RoboDK station: M20_v48.rdk

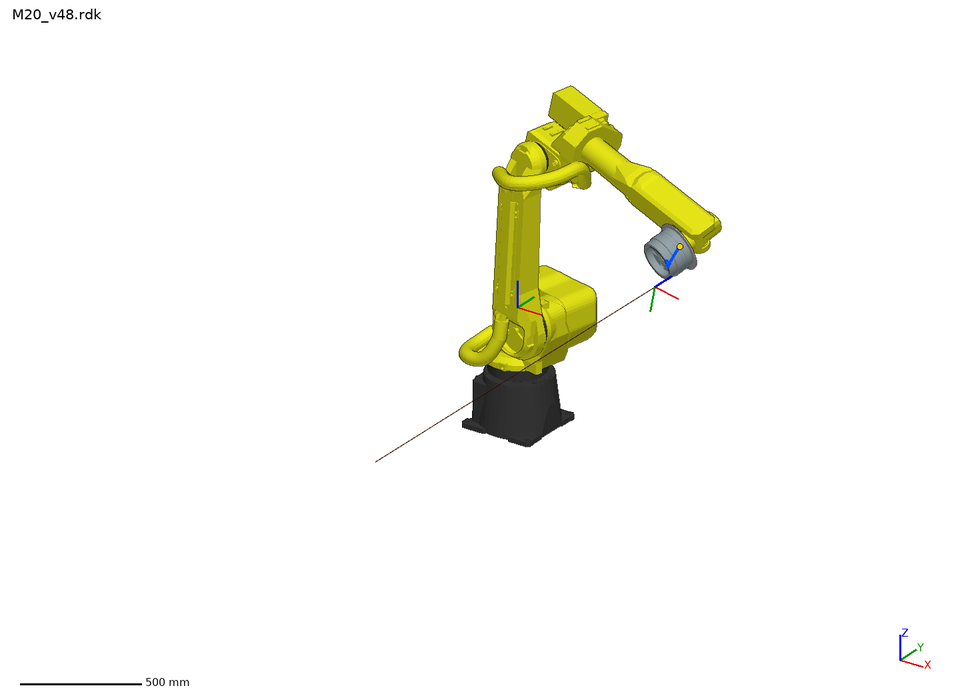
[picture v0: the station drawn from its stored meshes, robots at their saved joint values, targets as dots, program paths as lines]
Station M20_v48 (saved by RoboDK 5.2.2). Poses are relative to the parent item; angles as X-Y-Z fixed-axis rotations.
Station parameters (name, value as stored): CollisionFreePlanner, Fanuc M-20iA/35M, CollisionFreePlanner-Rob Fanuc M-20iA/35M
  - frame Fanuc M-20iA/35M Base at (0, 0, 525) mm
    - frame LASER_RTCP at (1000.3, -445, 552.3) mm, rotated rx -90 ry 10.19 rz 0 deg
      - object LASER_CAD at (0, 0, -1005) mm, size 2 x 2 x 2000 mm, geometry from laser.stl
    - robot Fanuc M-20iA/35M: 6 axes, payload 35 kg, reach 1813 mm, repeatability 0.04 mm, weight 252 kg
        modified DH rows (alpha deg, a mm, theta deg, d mm): 0, 0, 0, 525; -90, 150, -90, 0; 0, 790, 0, 0; -90, 150, 0, 860; 90, 0, 0, 0; -90, 0, 0, 100
        base shift (0, 0, -525) mm
        joint limits [-185, -110, -85, -200, -190, -450] to [185, 110, 245, 200, 190, 450]; home [0, 0, 0, 0, 0, 0]; saved at [-11.342, 3.915, -14.311, 70.129, -92.08, -387.18]
      - tool DIECAST, TCP at (0, 0, 200) mm, size 185 x 185 x 115 mm, geometry from B2 62-24 3naka.stp
      - tool Diecast15, TCP at (0, 0, 0) mm, geometry from I Co
      - tool holder_cylinder, TCP at (0, 0, 200) mm, size 220 x 220 x 5 mm, geometry from holder_cylinder.stl
  - machining project Diecast15 Settings: rotZ(0) | rotX(0)*rotY(0) | onStart | onPathStart | onApproach | onPoint | onRetract | onFinish | SetRPM(%1) | SetTool(%1) | Extruder(%1) | default | default | OutOnMov(%1) | OutOffMov(%1) | onPathFinish | M_RunCode(%1)
  - program Diecast15 (465 instructions, listed below)
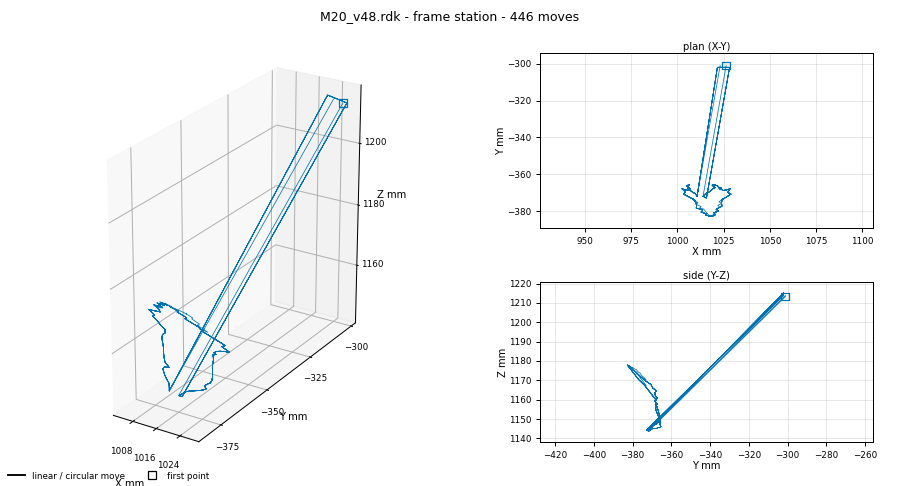
[picture p0: tool path of M20_v48.rdk in frame station, 446 of 446 moves have a stored position in this frame; points joined in program order, loops and branches not executed]

--- program Diecast15 (robot Fanuc M-20iA/35M) ---
  Smooth(1)
  Set speed (50.0 mm/s)
  Set Ref.: LASER_RTCP
  Set Tool: Diecast15
  Show Diecast15
  MoveJ 1 to (1.63, -138.5, 143.91) mm, rotated rx -165.35 ry -21.88 rz 21.81 deg; joints [-11.825, 0.745, -13.905, 69.881, -63.946, 28.2]
  MoveL 2 to (1.63, -138.5, 143.91) mm, rotated rx -165.35 ry -21.88 rz 21.81 deg; joints [-11.825, 0.745, -13.905, 69.881, -63.946, 28.2]
  MoveL 3 to (1.63, -67.79, 73.2) mm, rotated rx -165.35 ry -21.88 rz 21.81 deg; joints [-15.798, 1.644, -18.484, 72.688, -58.86, 24.658]
  MoveL 4 to (1.63, -67.79, 73.2) mm, rotated rx -165.35 ry -21.88 rz 21.81 deg; joints [-15.798, 1.644, -18.484, 72.688, -58.86, 24.658]
  Set speed (10.0 mm/s)
  MoveL 5 to (2.07, -68.2, 73.76) mm, rotated rx -165.47 ry -21.99 rz 21.64 deg; joints [-15.768, 1.64, -18.47, 72.794, -58.687, 24.483]
  MoveL 6 to (2.53, -68.64, 74.3) mm, rotated rx -165.57 ry -22.1 rz 21.49 deg; joints [-15.738, 1.639, -18.452, 72.873, -58.521, 24.337]
  MoveL 7 to (3.06, -69.11, 74.82) mm, rotated rx -165.64 ry -22.21 rz 21.37 deg; joints [-15.708, 1.647, -18.431, 72.918, -58.387, 24.236]
  MoveL 8 to (4.19, -69.63, 75.26) mm, rotated rx -165.57 ry -22.14 rz 21.47 deg; joints [-15.663, 1.734, -18.403, 72.823, -58.562, 24.363]
  MoveL 9 to (5.25, -69.87, 75.97) mm, rotated rx -165.69 ry -21.9 rz 21.48 deg; joints [-15.595, 1.808, -18.422, 73.065, -58.781, 24.144]
  MoveL 10 to (6.16, -70.02, 76.76) mm, rotated rx -165.89 ry -21.66 rz 21.42 deg; joints [-15.526, 1.864, -18.454, 73.413, -58.948, 23.797]
  MoveL 11 to (6.84, -70.15, 77.58) mm, rotated rx -166.69 ry -23.17 rz 23.41 deg; joints [-15.529, 1.8, -18.399, 72.916, -58.015, 26.249]
  MoveL 12 to (7.69, -70.84, 77.79) mm, rotated rx -166.55 ry -23.35 rz 23.41 deg; joints [-15.514, 1.85, -18.34, 72.636, -57.944, 26.482]
  MoveL 13 to (6.15, -70.44, 79.2) mm, rotated rx -167.55 ry -23.65 rz 22.5 deg; joints [-15.485, 1.581, -18.448, 73.906, -56.916, 24.951]
  MoveL 14 to (6.63, -71.02, 79.57) mm, rotated rx -167.55 ry -23.88 rz 22.37 deg; joints [-15.471, 1.583, -18.407, 73.817, -56.696, 24.96]
  MoveL 15 to (7.97, -72.41, 79.13) mm, rotated rx -166.89 ry -24.33 rz 22.62 deg; joints [-15.496, 1.704, -18.238, 72.683, -56.704, 26.052]
  MoveL 16 to (8.34, -73.51, 79.04) mm, rotated rx -166.59 ry -24.9 rz 22.52 deg; joints [-15.528, 1.7, -18.115, 72.031, -56.302, 26.565]
  MoveL 17 to (8.5, -74.86, 78.73) mm, rotated rx -166.17 ry -25.7 rz 22.39 deg; joints [-15.588, 1.674, -17.952, 71.101, -55.743, 27.309]
  MoveL 18 to (8.44, -76.15, 78.49) mm, rotated rx -166.38 ry -28.16 rz 24.17 deg; joints [-15.723, 1.552, -17.704, 69.121, -54.238, 30.819]
  MoveL 19 to (8.5, -77.42, 78.01) mm, rotated rx -165.94 ry -28.95 rz 23.91 deg; joints [-15.798, 1.526, -17.548, 68.152, -53.692, 31.516]
  MoveL 20 to (8.57, -78.66, 77.54) mm, rotated rx -165.5 ry -29.73 rz 23.67 deg; joints [-15.871, 1.503, -17.397, 67.191, -53.168, 32.216]
  MoveL 21 to (8.69, -79.8, 77.16) mm, rotated rx -165.12 ry -30.43 rz 23.43 deg; joints [-15.935, 1.485, -17.262, 66.331, -52.694, 32.845]
  MoveL 22 to (8.83, -80.8, 76.93) mm, rotated rx -164.84 ry -31.04 rz 23.21 deg; joints [-15.986, 1.466, -17.149, 65.628, -52.254, 33.35]
  MoveL 23 to (8.86, -81.65, 76.86) mm, rotated rx -164.67 ry -31.59 rz 22.95 deg; joints [-16.027, 1.43, -17.059, 65.109, -51.784, 33.692]
  MoveL 24 to (8.62, -82.36, 76.99) mm, rotated rx -164.65 ry -32.12 rz 22.64 deg; joints [-16.061, 1.358, -16.994, 64.807, -51.211, 33.829]
  MoveL 25 to (8.14, -82.88, 77.34) mm, rotated rx -164.81 ry -32.62 rz 22.28 deg; joints [-16.085, 1.251, -16.958, 64.762, -50.545, 33.726]
  MoveL 26 to (8.9, -83.1, 77.88) mm, rotated rx -164.95 ry -32.61 rz 22.32 deg; joints [-16.042, 1.287, -16.962, 64.907, -50.532, 33.64]
  MoveL 27 to (8.4, -83.82, 77.16) mm, rotated rx -163.11 ry -28.11 rz 16.62 deg; joints [-15.881, 1.436, -17.144, 68.063, -52.662, 25.505]
  MoveL 28 to (9.59, -85.18, 76.37) mm, rotated rx -162.32 ry -28.55 rz 16.51 deg; joints [-15.938, 1.548, -16.98, 66.869, -52.596, 26.417]
  MoveL 29 to (10.68, -85.68, 76.53) mm, rotated rx -162.2 ry -28.63 rz 16.49 deg; joints [-15.918, 1.623, -16.944, 66.673, -52.606, 26.556]
  MoveL 30 to (11.92, -86.02, 76.84) mm, rotated rx -162.17 ry -28.58 rz 16.53 deg; joints [-15.879, 1.713, -16.933, 66.641, -52.715, 26.587]
  MoveL 31 to (13.25, -86.21, 77.3) mm, rotated rx -162.25 ry -28.48 rz 16.65 deg; joints [-15.826, 1.808, -16.941, 66.743, -52.87, 26.562]
  MoveL 32 to (11.52, -88.17, 75.33) mm, rotated rx -160.24 ry -19.61 rz 6.74 deg; joints [-15.594, 2.135, -17.19, 71.435, -57.463, 12.158]
  MoveL 33 to (13.08, -89.68, 74.39) mm, rotated rx -159.35 ry -19.76 rz 6.39 deg; joints [-15.647, 2.276, -17.02, 70.374, -57.388, 12.626]
  MoveL 34 to (7.41, -92.83, 71.24) mm, rotated rx -160.05 ry -2.49 rz -10.95 deg; joints [-15.35, 3.01, -17.298, 75.065, -67.641, -11.935]
  MoveL 35 to (6.99, -94.6, 69.39) mm, rotated rx -158.65 ry -2.96 rz -11.41 deg; joints [-15.51, 2.946, -17.033, 73.655, -66.695, -11.359]
  MoveL 36 to (7.01, -96.01, 67.92) mm, rotated rx -157.53 ry -3.3 rz -11.74 deg; joints [-15.633, 2.926, -16.826, 72.509, -66.001, -10.847]
  MoveL 37 to (3.4, -97.81, 66.12) mm, rotated rx -158.66 ry 3.54 rz -19.31 deg; joints [-15.646, 3.148, -16.736, 72.608, -69.699, -20.384]
  MoveL 38 to (4.11, -98.25, 65.89) mm, rotated rx -158.38 ry 3.45 rz -19.41 deg; joints [-15.66, 3.182, -16.686, 72.348, -69.482, -20.301]
  MoveL 39 to (4.55, -99.05, 65.14) mm, rotated rx -157.76 ry 3.32 rz -19.55 deg; joints [-15.718, 3.197, -16.575, 71.749, -69.084, -20.047]
  MoveL 40 to (1.71, -100.01, 64.3) mm, rotated rx -159.5 ry 8.48 rz -25.55 deg; joints [-15.716, 3.361, -16.523, 71.702, -71.957, -27.421]
  MoveL 41 to (2.18, -100.59, 63.71) mm, rotated rx -159 ry 8.39 rz -25.68 deg; joints [-15.76, 3.374, -16.441, 71.262, -71.59, -27.288]
  MoveL 42 to (2.6, -101.12, 63.22) mm, rotated rx -158.54 ry 8.27 rz -25.84 deg; joints [-15.799, 3.378, -16.368, 70.876, -71.207, -27.191]
  MoveL 43 to (0.07, -101.65, 62.81) mm, rotated rx -160.41 ry 12.13 rz -30.92 deg; joints [-15.802, 3.467, -16.33, 70.757, -73.31, -33.152]
  MoveL 44 to (0.46, -101.9, 62.5) mm, rotated rx -160.1 ry 12.01 rz -31.1 deg; joints [-15.827, 3.465, -16.29, 70.542, -72.966, -33.17]
  MoveL 45 to (0.93, -102.06, 62.36) mm, rotated rx -159.88 ry 11.87 rz -31.27 deg; joints [-15.838, 3.467, -16.268, 70.431, -72.668, -33.226]
  MoveL 46 to (-1.4, -102.13, 62.39) mm, rotated rx -162.06 ry 15.05 rz -36.05 deg; joints [-15.824, 3.527, -16.27, 70.42, -74.51, -38.652]
  MoveL 47 to (-0.93, -102.06, 62.36) mm, rotated rx -161.94 ry 14.86 rz -36.23 deg; joints [-15.826, 3.525, -16.275, 70.43, -74.216, -38.774]
  MoveL 48 to (-0.46, -101.91, 62.5) mm, rotated rx -161.88 ry 14.62 rz -36.44 deg; joints [-15.816, 3.516, -16.296, 70.541, -73.922, -38.94]
  MoveL 49 to (-3.14, -101.52, 62.94) mm, rotated rx -164.88 ry 17.8 rz -42.05 deg; joints [-15.783, 3.572, -16.337, 70.604, -76.011, -45.083]
  MoveL 50 to (-2.61, -101.12, 63.22) mm, rotated rx -164.89 ry 17.45 rz -42.26 deg; joints [-15.762, 3.559, -16.388, 70.854, -75.702, -45.295]
  MoveL 51 to (-2.18, -100.59, 63.71) mm, rotated rx -164.95 ry 16.98 rz -42.5 deg; joints [-15.729, 3.524, -16.458, 71.232, -75.342, -45.573]
  MoveL 52 to (-5.22, -99.67, 64.64) mm, rotated rx -169.38 ry 20.42 rz -49.8 deg; joints [-15.671, 3.63, -16.54, 71.222, -78.128, -53.168]
  MoveL 53 to (-4.55, -99.05, 65.14) mm, rotated rx -169.47 ry 19.97 rz -49.94 deg; joints [-15.63, 3.626, -16.624, 71.633, -77.889, -53.393]
  MoveL 54 to (-4.11, -98.25, 65.89) mm, rotated rx -169.57 ry 19.34 rz -50.15 deg; joints [-15.578, 3.582, -16.731, 72.2, -77.538, -53.711]
  MoveL 55 to (-7.39, -97.12, 66.82) mm, rotated rx -176.04 ry 23.25 rz -59.97 deg; joints [-15.54, 3.829, -16.77, 71.378, -81.442, -63.181]
  MoveL 56 to (-7.01, -96.01, 67.92) mm, rotated rx -176.09 ry 22.37 rz -60.15 deg; joints [-15.463, 3.763, -16.921, 72.174, -81.052, -63.577]
  MoveL 57 to (-7, -94.6, 69.39) mm, rotated rx -176.12 ry 21.21 rz -60.42 deg; joints [-15.371, 3.636, -17.112, 73.215, -80.491, -64.129]
  MoveL 58 to (-7.48, -92.8, 71.26) mm, rotated rx -176.27 ry 19.82 rz -61.04 deg; joints [-15.262, 3.451, -17.348, 74.505, -79.855, -65.095]
  MoveL 59 to (-13.13, -89.63, 74.43) mm, rotated rx 165.84 ry 24.86 rz -85.39 deg; joints [-15.239, 4.306, -17.25, 69.785, -89.701, -86.616]
  MoveL 60 to (-11.56, -88.14, 75.37) mm, rotated rx 165.82 ry 24 rz -85.44 deg; joints [-15.148, 4.371, -17.444, 70.572, -89.67, -87.094]
  MoveL 61 to (-13.24, -86.21, 77.29) mm, rotated rx 156.15 ry 23.72 rz -98.23 deg; joints [-15.214, 4.82, -17.286, 66.859, -93.953, -98.196]
  MoveL 62 to (-11.92, -86.02, 76.84) mm, rotated rx 156.02 ry 23.8 rz -98.23 deg; joints [-15.224, 4.938, -17.301, 66.771, -94.063, -98.181]
  MoveL 63 to (-10.68, -85.68, 76.53) mm, rotated rx 155.96 ry 23.78 rz -98.19 deg; joints [-15.223, 5.038, -17.334, 66.788, -94.12, -98.189]
  MoveL 64 to (-9.59, -85.18, 76.37) mm, rotated rx 156.03 ry 23.66 rz -98.13 deg; joints [-15.212, 5.11, -17.387, 66.917, -94.088, -98.228]
  MoveL 65 to (-8.43, -83.79, 77.19) mm, rotated rx 156.12 ry 22.88 rz -98.07 deg; joints [-15.132, 5.162, -17.564, 67.624, -94.128, -98.634]
  MoveL 66 to (-8.89, -83.12, 77.86) mm, rotated rx 151.43 ry 22.02 rz -104.29 deg; joints [-15.2, 5.396, -17.434, 65.454, -96.039, -104.222]
  MoveL 67 to (-8.17, -82.86, 77.3) mm, rotated rx 151.41 ry 22.13 rz -104.41 deg; joints [-15.224, 5.452, -17.438, 65.321, -95.957, -104.272]
  MoveL 68 to (-8.66, -82.3, 76.95) mm, rotated rx 151.99 ry 22.19 rz -104.66 deg; joints [-15.244, 5.337, -17.453, 65.339, -95.242, -104.451]
  MoveL 69 to (-8.87, -81.54, 76.84) mm, rotated rx 152.59 ry 22.08 rz -104.73 deg; joints [-15.242, 5.245, -17.508, 65.555, -94.631, -104.594]
  MoveL 70 to (-8.81, -80.61, 76.95) mm, rotated rx 153.19 ry 21.82 rz -104.65 deg; joints [-15.22, 5.176, -17.596, 65.942, -94.124, -104.708]
  MoveL 71 to (-8.67, -79.52, 77.23) mm, rotated rx 153.85 ry 21.44 rz -104.48 deg; joints [-15.183, 5.108, -17.712, 66.479, -93.638, -104.817]
  MoveL 72 to (-8.55, -78.28, 77.67) mm, rotated rx 154.6 ry 20.95 rz -104.25 deg; joints [-15.134, 5.029, -17.851, 67.141, -93.121, -104.939]
  MoveL 73 to (-8.49, -76.94, 78.18) mm, rotated rx 155.41 ry 20.4 rz -104 deg; joints [-15.081, 4.938, -18.004, 67.878, -92.57, -105.079]
  MoveL 74 to (-8.51, -75.85, 78.43) mm, rotated rx 157.93 ry 20.23 rz -101.5 deg; joints [-15.019, 4.733, -18.19, 69.315, -91.216, -103.146]
  MoveL 75 to (-8.47, -74.37, 78.86) mm, rotated rx 158.81 ry 19.62 rz -101.14 deg; joints [-14.972, 4.635, -18.36, 70.138, -90.615, -103.216]
  MoveL 76 to (-8.24, -73.1, 79.09) mm, rotated rx 159.5 ry 19.14 rz -100.87 deg; joints [-14.939, 4.574, -18.501, 70.788, -90.141, -103.29]
  MoveL 77 to (-7.81, -72.09, 79.1) mm, rotated rx 159.97 ry 18.82 rz -100.7 deg; joints [-14.922, 4.553, -18.608, 71.229, -89.799, -103.36]
  MoveL 78 to (-6.43, -70.76, 79.48) mm, rotated rx 160.25 ry 18.17 rz -100.09 deg; joints [-14.863, 4.638, -18.793, 72.015, -89.896, -103.231]
  MoveL 79 to (-7.32, -70.96, 78.29) mm, rotated rx 160.6 ry 18.8 rz -100.96 deg; joints [-14.957, 4.51, -18.675, 71.344, -89.033, -103.65]
  MoveL 80 to (-7.42, -70.56, 77.72) mm, rotated rx 160.97 ry 18.94 rz -101.27 deg; joints [-14.993, 4.451, -18.675, 71.246, -88.491, -103.87]
  MoveL 81 to (-6.7, -70.14, 77.26) mm, rotated rx 162.83 ry 19.1 rz -98.92 deg; joints [-14.989, 4.376, -18.762, 72.009, -87.526, -101.813]
  MoveL 82 to (-5.92, -69.96, 76.53) mm, rotated rx 162.68 ry 19.31 rz -99.12 deg; joints [-15.024, 4.453, -18.75, 71.753, -87.526, -101.899]
  MoveL 83 to (-5.02, -69.82, 75.79) mm, rotated rx 162.46 ry 19.53 rz -99.3 deg; joints [-15.058, 4.549, -18.737, 71.479, -87.597, -101.964]
  MoveL 84 to (-3.99, -69.56, 75.15) mm, rotated rx 162.26 ry 19.65 rz -99.38 deg; joints [-15.082, 4.654, -18.745, 71.312, -87.717, -101.987]
  MoveL 85 to (-2.94, -69.02, 74.77) mm, rotated rx 162.21 ry 19.58 rz -99.26 deg; joints [-15.086, 4.746, -18.799, 71.398, -87.801, -101.959]
  MoveL 86 to (-2.49, -68.6, 74.25) mm, rotated rx 162.34 ry 19.64 rz -99.39 deg; joints [-15.11, 4.765, -18.817, 71.348, -87.59, -102.065]
  MoveL 87 to (-2.05, -68.18, 73.73) mm, rotated rx 162.47 ry 19.7 rz -99.53 deg; joints [-15.134, 4.782, -18.835, 71.298, -87.37, -102.174]
  MoveL 88 to (-1.64, -67.79, 73.2) mm, rotated rx 162.63 ry 19.79 rz -99.64 deg; joints [-15.159, 4.794, -18.85, 71.241, -87.124, -102.251]
  Set speed (50.0 mm/s)
  MoveL 89 to (-1.64, -67.79, 73.2) mm, rotated rx 162.63 ry 19.79 rz -99.64 deg; joints [-15.159, 4.794, -18.85, 71.241, -87.124, -102.251]
  MoveL 90 to (-3.35, -139.46, 142.95) mm, rotated rx -174.85 ry 17.93 rz -70.52 deg; joints [-11.389, 2.134, -14.376, 73.889, -79.145, -72.161]
  Set speed (50.0 mm/s)
  MoveL 91 to (3.35, -139.46, 142.95) mm, rotated rx -173.27 ry 17.41 rz -71.64 deg; joints [-11.355, 2.358, -14.405, 73.913, -77.143, -73.209]
  MoveL 92 to (3.35, -68.75, 72.24) mm, rotated rx -173.27 ry 17.41 rz -71.64 deg; joints [-15.25, 3.252, -18.966, 75.969, -72.353, -76.766]
  MoveL 93 to (1.63, -67.79, 73.2) mm, rotated rx -154.57 ry 6.2 rz -45.94 deg; joints [-15.798, 1.644, -18.484, 72.688, -58.86, -47.342]
  Set speed (10.0 mm/s)
  MoveL 94 to (2.07, -68.2, 73.76) mm, rotated rx -154.51 ry 6.06 rz -46.15 deg; joints [-15.768, 1.64, -18.47, 72.794, -58.687, -47.517]
  MoveL 95 to (2.53, -68.64, 74.3) mm, rotated rx -154.43 ry 5.93 rz -46.33 deg; joints [-15.738, 1.639, -18.452, 72.873, -58.521, -47.663]
  MoveL 96 to (3.06, -69.11, 74.82) mm, rotated rx -154.36 ry 5.83 rz -46.47 deg; joints [-15.708, 1.647, -18.431, 72.918, -58.387, -47.764]
  MoveL 97 to (4.19, -69.63, 75.26) mm, rotated rx -154.4 ry 5.92 rz -46.34 deg; joints [-15.663, 1.734, -18.403, 72.823, -58.562, -47.637]
  MoveL 98 to (5.25, -69.87, 75.97) mm, rotated rx -154.66 ry 5.9 rz -46.41 deg; joints [-15.595, 1.808, -18.422, 73.065, -58.781, -47.856]
  MoveL 99 to (6.16, -70.02, 76.76) mm, rotated rx -154.96 ry 5.82 rz -46.57 deg; joints [-15.526, 1.864, -18.454, 73.413, -58.948, -48.203]
  MoveL 100 to (6.84, -70.15, 77.58) mm, rotated rx -153.84 ry 4.57 rz -44.78 deg; joints [-15.529, 1.8, -18.399, 72.916, -58.015, -45.751]
  MoveL 101 to (7.69, -70.84, 77.79) mm, rotated rx -153.61 ry 4.62 rz -44.71 deg; joints [-15.514, 1.85, -18.34, 72.636, -57.944, -45.518]
  MoveL 102 to (6.15, -70.44, 79.2) mm, rotated rx -153.67 ry 3.66 rz -46.03 deg; joints [-15.485, 1.581, -18.448, 73.906, -56.916, -47.049]
  MoveL 103 to (6.63, -71.02, 79.57) mm, rotated rx -153.47 ry 3.58 rz -46.14 deg; joints [-15.471, 1.583, -18.407, 73.817, -56.696, -47.039]
  MoveL 104 to (7.97, -72.41, 79.13) mm, rotated rx -152.82 ry 3.98 rz -45.58 deg; joints [-15.496, 1.704, -18.238, 72.683, -56.704, -45.948]
  MoveL 105 to (8.34, -73.51, 79.04) mm, rotated rx -152.19 ry 4.01 rz -45.51 deg; joints [-15.528, 1.7, -18.115, 72.031, -56.302, -45.435]
  MoveL 106 to (8.5, -74.86, 78.73) mm, rotated rx -151.3 ry 4.06 rz -45.4 deg; joints [-15.588, 1.674, -17.952, 71.101, -55.743, -44.691]
  MoveL 107 to (8.44, -76.15, 78.49) mm, rotated rx -149.09 ry 2.96 rz -43.59 deg; joints [-15.723, 1.552, -17.704, 69.121, -54.238, -41.181]
  MoveL 108 to (8.5, -77.42, 78.01) mm, rotated rx -148.21 ry 3.01 rz -43.58 deg; joints [-15.798, 1.526, -17.548, 68.152, -53.692, -40.484]
  MoveL 109 to (8.57, -78.66, 77.54) mm, rotated rx -147.35 ry 3.07 rz -43.57 deg; joints [-15.871, 1.503, -17.397, 67.191, -53.168, -39.784]
  MoveL 110 to (8.69, -79.8, 77.16) mm, rotated rx -146.58 ry 3.1 rz -43.57 deg; joints [-15.935, 1.485, -17.262, 66.331, -52.694, -39.155]
  MoveL 111 to (8.83, -80.8, 76.93) mm, rotated rx -145.92 ry 3.09 rz -43.61 deg; joints [-15.986, 1.466, -17.149, 65.628, -52.254, -38.65]
  MoveL 112 to (8.86, -81.65, 76.86) mm, rotated rx -145.35 ry 3 rz -43.75 deg; joints [-16.027, 1.43, -17.059, 65.109, -51.784, -38.308]
  MoveL 113 to (8.62, -82.36, 76.99) mm, rotated rx -144.85 ry 2.8 rz -44.03 deg; joints [-16.061, 1.358, -16.994, 64.807, -51.211, -38.171]
  MoveL 114 to (8.14, -82.88, 77.34) mm, rotated rx -144.45 ry 2.48 rz -44.46 deg; joints [-16.085, 1.251, -16.958, 64.762, -50.545, -38.274]
  MoveL 115 to (8.9, -83.1, 77.88) mm, rotated rx -144.51 ry 2.38 rz -44.5 deg; joints [-16.042, 1.287, -16.962, 64.907, -50.532, -38.36]
  MoveL 116 to (8.4, -83.82, 77.16) mm, rotated rx -148 ry 5.63 rz -49.51 deg; joints [-15.881, 1.436, -17.144, 68.063, -52.662, -46.495]
  MoveL 117 to (9.59, -85.18, 76.37) mm, rotated rx -147.32 ry 6.08 rz -49.17 deg; joints [-15.938, 1.548, -16.98, 66.869, -52.596, -45.583]
  MoveL 118 to (10.68, -85.68, 76.53) mm, rotated rx -147.2 ry 6.15 rz -49.13 deg; joints [-15.918, 1.623, -16.944, 66.673, -52.606, -45.444]
  MoveL 119 to (11.92, -86.02, 76.84) mm, rotated rx -147.23 ry 6.19 rz -49.07 deg; joints [-15.879, 1.713, -16.933, 66.641, -52.715, -45.413]
  MoveL 120 to (13.25, -86.21, 77.3) mm, rotated rx -147.36 ry 6.17 rz -49 deg; joints [-15.826, 1.808, -16.941, 66.743, -52.87, -45.438]
  MoveL 121 to (11.52, -88.17, 75.33) mm, rotated rx -154.78 ry 11.49 rz -59.23 deg; joints [-15.594, 2.135, -17.19, 71.435, -57.463, -59.842]
  MoveL 122 to (13.08, -89.68, 74.39) mm, rotated rx -154.29 ry 12.19 rz -59.18 deg; joints [-15.647, 2.276, -17.02, 70.374, -57.388, -59.374]
  MoveL 123 to (7.41, -92.83, 71.24) mm, rotated rx -171.12 ry 18.11 rz -81.1 deg; joints [-15.35, 3.01, -17.298, 75.065, -67.641, -83.935]
  MoveL 124 to (6.99, -94.6, 69.39) mm, rotated rx -170.15 ry 19.26 rz -81.18 deg; joints [-15.51, 2.946, -17.033, 73.655, -66.695, -83.358]
  MoveL 125 to (7.01, -96.01, 67.92) mm, rotated rx -169.4 ry 20.18 rz -81.19 deg; joints [-15.633, 2.926, -16.826, 72.509, -66.001, -82.847]
  MoveL 126 to (3.4, -97.81, 66.12) mm, rotated rx -176.71 ry 21.38 rz -91.36 deg; joints [-15.646, 3.148, -16.736, 72.608, -69.699, -92.384]
  MoveL 127 to (4.11, -98.25, 65.89) mm, rotated rx -176.52 ry 21.62 rz -91.41 deg; joints [-15.66, 3.182, -16.686, 72.348, -69.482, -92.301]
  MoveL 128 to (4.55, -99.05, 65.14) mm, rotated rx -176.18 ry 22.17 rz -91.45 deg; joints [-15.718, 3.197, -16.575, 71.749, -69.084, -92.047]
  MoveL 129 to (1.71, -100.01, 64.3) mm, rotated rx 177.95 ry 22.02 rz -99.48 deg; joints [-15.716, 3.361, -16.523, 71.702, -71.957, -99.421]
  MoveL 130 to (2.18, -100.59, 63.71) mm, rotated rx 178.19 ry 22.47 rz -99.6 deg; joints [-15.76, 3.374, -16.441, 71.262, -71.59, -99.288]
  MoveL 131 to (2.6, -101.12, 63.22) mm, rotated rx 178.45 ry 22.88 rz -99.73 deg; joints [-15.799, 3.378, -16.368, 70.876, -71.208, -99.191]
  MoveL 132 to (0.07, -101.65, 62.81) mm, rotated rx 173.89 ry 22.13 rz -106.22 deg; joints [-15.802, 3.467, -16.33, 70.757, -73.31, -105.152]
  MoveL 133 to (0.46, -101.9, 62.5) mm, rotated rx 174.1 ry 22.4 rz -106.38 deg; joints [-15.827, 3.465, -16.29, 70.542, -72.966, -105.17]
  MoveL 134 to (0.93, -102.06, 62.36) mm, rotated rx 174.3 ry 22.56 rz -106.52 deg; joints [-15.838, 3.467, -16.268, 70.431, -72.668, -105.226]
  MoveL 135 to (-1.4, -102.13, 62.39) mm, rotated rx 170.42 ry 21.29 rz -112.24 deg; joints [-15.824, 3.527, -16.27, 70.42, -74.51, -110.652]
  MoveL 136 to (-0.93, -102.06, 62.36) mm, rotated rx 170.65 ry 21.36 rz -112.38 deg; joints [-15.826, 3.525, -16.275, 70.43, -74.216, -110.774]
  MoveL 137 to (-3.73, -99.39, 66.32) mm, rotated rx 173.02 ry 19.79 rz -112.85 deg; joints [-15.645, 2.973, -16.65, 72.928, -72.46, -112.562]
  MoveL 138 to (-5.81, -98.78, 66.97) mm, rotated rx 169.22 ry 17.82 rz -118.67 deg; joints [-15.581, 3.077, -16.727, 73.108, -74.694, -118.451]
  MoveL 139 to (-5.31, -98.38, 67.24) mm, rotated rx 169.58 ry 17.74 rz -118.77 deg; joints [-15.562, 3.063, -16.778, 73.365, -74.386, -118.687]
  MoveL 140 to (-4.91, -97.85, 67.7) mm, rotated rx 170.03 ry 17.58 rz -118.88 deg; joints [-15.533, 3.029, -16.847, 73.743, -74.034, -118.99]
  MoveL 141 to (-7.21, -96.71, 68.8) mm, rotated rx 165.64 ry 14.42 rz -125.83 deg; joints [-15.442, 3.207, -16.969, 73.837, -77.072, -126.355]
  MoveL 142 to (-6.57, -96.1, 69.26) mm, rotated rx 166.05 ry 14.25 rz -125.85 deg; joints [-15.406, 3.203, -17.051, 74.238, -76.839, -126.597]
  MoveL 143 to (-6.15, -95.3, 69.94) mm, rotated rx 166.63 ry 14.02 rz -125.9 deg; joints [-15.361, 3.162, -17.156, 74.789, -76.503, -126.935]
  MoveL 144 to (-8.5, -93.99, 71.03) mm, rotated rx 161.23 ry 9.24 rz -134.4 deg; joints [-15.283, 3.514, -17.234, 74.035, -80.805, -136.218]
  MoveL 145 to (-8.16, -92.87, 72.03) mm, rotated rx 162.04 ry 8.98 rz -134.45 deg; joints [-15.216, 3.451, -17.383, 74.805, -80.432, -136.633]
  MoveL 146 to (-7, -94.6, 69.39) mm, rotated rx 160.76 ry 9.9 rz -134.83 deg; joints [-15.371, 3.636, -17.112, 73.215, -80.491, -136.129]
  MoveL 147 to (-7.48, -92.8, 71.26) mm, rotated rx 162.08 ry 9.38 rz -135.18 deg; joints [-15.262, 3.451, -17.348, 74.505, -79.855, -137.095]
  MoveL 148 to (-13.13, -89.63, 74.43) mm, rotated rx 151.97 ry -4.66 rz -153.08 deg; joints [-15.239, 4.306, -17.25, 69.785, -89.701, -158.616]
  MoveL 149 to (-11.56, -88.14, 75.37) mm, rotated rx 152.75 ry -5 rz -153.2 deg; joints [-15.148, 4.371, -17.444, 70.572, -89.67, -159.094]
  MoveL 150 to (-13.24, -86.21, 77.29) mm, rotated rx 149.31 ry -13.16 rz -161.52 deg; joints [-15.214, 4.82, -17.286, 66.859, -93.953, -170.196]
  MoveL 151 to (-11.92, -86.02, 76.84) mm, rotated rx 149.18 ry -13.24 rz -161.44 deg; joints [-15.224, 4.938, -17.301, 66.771, -94.063, -170.181]
  MoveL 152 to (-10.68, -85.68, 76.53) mm, rotated rx 149.18 ry -13.29 rz -161.38 deg; joints [-15.223, 5.038, -17.334, 66.788, -94.12, -170.188]
  MoveL 153 to (-9.59, -85.18, 76.37) mm, rotated rx 149.31 ry -13.29 rz -161.38 deg; joints [-15.212, 5.11, -17.387, 66.917, -94.088, -170.228]
  MoveL 154 to (-8.43, -83.79, 77.19) mm, rotated rx 150.07 ry -13.56 rz -161.53 deg; joints [-15.132, 5.162, -17.564, 67.623, -94.128, -170.634]
  MoveL 155 to (-8.89, -83.12, 77.86) mm, rotated rx 148.77 ry -17.81 rz -165.61 deg; joints [-15.2, 5.396, -17.434, 65.454, -96.039, -176.222]
  MoveL 156 to (-8.17, -82.86, 77.3) mm, rotated rx 148.66 ry -17.77 rz -165.68 deg; joints [-15.224, 5.452, -17.438, 65.321, -95.958, -176.272]
  MoveL 157 to (-8.66, -82.3, 76.95) mm, rotated rx 148.88 ry -17.27 rz -166.21 deg; joints [-15.244, 5.337, -17.453, 65.339, -95.242, -176.451]
  MoveL 158 to (-8.87, -81.54, 76.84) mm, rotated rx 149.25 ry -16.83 rz -166.62 deg; joints [-15.242, 5.245, -17.508, 65.555, -94.631, -176.594]
  MoveL 159 to (-8.81, -80.61, 76.95) mm, rotated rx 149.77 ry -16.46 rz -166.92 deg; joints [-15.22, 5.176, -17.596, 65.942, -94.124, -176.708]
  MoveL 160 to (-8.67, -79.52, 77.23) mm, rotated rx 150.42 ry -16.09 rz -167.17 deg; joints [-15.183, 5.108, -17.712, 66.479, -93.638, -176.817]
  MoveL 161 to (-8.55, -78.28, 77.67) mm, rotated rx 151.2 ry -15.69 rz -167.42 deg; joints [-15.134, 5.029, -17.851, 67.141, -93.121, -176.938]
  MoveL 162 to (-8.49, -76.94, 78.18) mm, rotated rx 152.05 ry -15.26 rz -167.68 deg; joints [-15.081, 4.938, -18.004, 67.878, -92.57, -177.079]
  MoveL 163 to (-8.51, -75.85, 78.43) mm, rotated rx 153.28 ry -13.21 rz -166.36 deg; joints [-15.019, 4.733, -18.19, 69.315, -91.216, -175.146]
  MoveL 164 to (-8.47, -74.37, 78.86) mm, rotated rx 154.2 ry -12.71 rz -166.51 deg; joints [-14.972, 4.635, -18.36, 70.138, -90.615, -175.216]
  MoveL 165 to (-8.24, -73.1, 79.09) mm, rotated rx 154.92 ry -12.32 rz -166.63 deg; joints [-14.939, 4.574, -18.501, 70.788, -90.141, -175.29]
  MoveL 166 to (-7.81, -72.09, 79.1) mm, rotated rx 155.41 ry -12.05 rz -166.72 deg; joints [-14.922, 4.553, -18.608, 71.229, -89.799, -175.36]
  MoveL 167 to (-6.43, -70.76, 79.48) mm, rotated rx 156.13 ry -12.07 rz -166.34 deg; joints [-14.863, 4.638, -18.793, 72.015, -89.896, -175.231]
  MoveL 168 to (-7.32, -70.96, 78.29) mm, rotated rx 155.67 ry -11.5 rz -167.23 deg; joints [-14.957, 4.51, -18.675, 71.344, -89.033, -175.65]
  MoveL 169 to (-7.42, -70.56, 77.72) mm, rotated rx 155.69 ry -11.13 rz -167.67 deg; joints [-14.993, 4.451, -18.675, 71.246, -88.491, -175.87]
  MoveL 170 to (-6.7, -70.14, 77.26) mm, rotated rx 156.24 ry -9.45 rz -166.02 deg; joints [-14.989, 4.376, -18.762, 72.009, -87.526, -173.813]
  MoveL 171 to (-5.92, -69.96, 76.53) mm, rotated rx 155.99 ry -9.5 rz -166.12 deg; joints [-15.024, 4.453, -18.75, 71.754, -87.526, -173.899]
  MoveL 172 to (-5.02, -69.82, 75.79) mm, rotated rx 155.71 ry -9.6 rz -166.19 deg; joints [-15.058, 4.549, -18.737, 71.479, -87.597, -173.964]
  MoveL 173 to (-3.99, -69.56, 75.15) mm, rotated rx 155.51 ry -9.73 rz -166.16 deg; joints [-15.082, 4.654, -18.745, 71.312, -87.717, -173.987]
  MoveL 174 to (-2.94, -69.02, 74.77) mm, rotated rx 155.56 ry -9.8 rz -166.04 deg; joints [-15.086, 4.746, -18.799, 71.398, -87.801, -173.959]
  MoveL 175 to (-2.49, -68.6, 74.25) mm, rotated rx 155.55 ry -9.67 rz -166.21 deg; joints [-15.11, 4.765, -18.817, 71.348, -87.59, -174.065]
  MoveL 176 to (-2.05, -68.18, 73.73) mm, rotated rx 155.54 ry -9.53 rz -166.39 deg; joints [-15.134, 4.782, -18.835, 71.298, -87.37, -174.174]
  MoveL 177 to (-1.64, -67.79, 73.2) mm, rotated rx 155.53 ry -9.36 rz -166.55 deg; joints [-15.159, 4.794, -18.85, 71.241, -87.124, -174.251]
  Set speed (50.0 mm/s)
  MoveL 178 to (-1.64, -67.79, 73.2) mm, rotated rx 155.53 ry -9.36 rz -166.55 deg; joints [-15.159, 4.794, -18.85, 71.241, -87.124, -174.251]
  MoveL 179 to (-3.35, -139.46, 142.95) mm, rotated rx 164.3 ry 10.15 rz -144.74 deg; joints [-11.389, 2.134, -14.376, 73.889, -79.145, -144.161]
  Set speed (50.0 mm/s)
  MoveL 180 to (3.35, -139.46, 142.95) mm, rotated rx 165.22 ry 11.47 rz -146.16 deg; joints [-11.355, 2.358, -14.405, 73.913, -77.143, -145.209]
  MoveL 181 to (3.35, -68.75, 72.24) mm, rotated rx 165.22 ry 11.47 rz -146.16 deg; joints [-15.25, 3.252, -18.966, 75.969, -72.353, -148.766]
  MoveL 182 to (1.63, -67.79, 73.2) mm, rotated rx -178.14 ry 26.07 rz -118.91 deg; joints [-15.798, 1.644, -18.484, 72.688, -58.86, -119.342]
  Set speed (10.0 mm/s)
  MoveL 183 to (2.07, -68.2, 73.76) mm, rotated rx -177.97 ry 26.08 rz -119.05 deg; joints [-15.768, 1.64, -18.47, 72.794, -58.687, -119.517]
  MoveL 184 to (2.53, -68.64, 74.3) mm, rotated rx -177.81 ry 26.12 rz -119.16 deg; joints [-15.738, 1.639, -18.452, 72.873, -58.521, -119.663]
  MoveL 185 to (3.06, -69.11, 74.82) mm, rotated rx -177.68 ry 26.16 rz -119.25 deg; joints [-15.708, 1.647, -18.431, 72.918, -58.387, -119.764]
  MoveL 186 to (4.19, -69.63, 75.26) mm, rotated rx -177.78 ry 26.14 rz -119.17 deg; joints [-15.663, 1.734, -18.403, 72.823, -58.563, -119.637]
  MoveL 187 to (5.25, -69.87, 75.97) mm, rotated rx -177.85 ry 25.89 rz -119.24 deg; joints [-15.595, 1.808, -18.422, 73.065, -58.781, -119.856]
  MoveL 188 to (6.16, -70.02, 76.76) mm, rotated rx -177.86 ry 25.58 rz -119.38 deg; joints [-15.526, 1.864, -18.454, 73.413, -58.948, -120.203]
  MoveL 189 to (6.84, -70.15, 77.58) mm, rotated rx -176.16 ry 26.27 rz -116.95 deg; joints [-15.529, 1.8, -18.399, 72.916, -58.015, -117.751]
  MoveL 190 to (7.69, -70.84, 77.79) mm, rotated rx -176.14 ry 26.5 rz -116.89 deg; joints [-15.514, 1.85, -18.34, 72.636, -57.944, -117.518]
  MoveL 191 to (6.15, -70.44, 79.2) mm, rotated rx -175.14 ry 26.15 rz -117.75 deg; joints [-15.485, 1.581, -18.448, 73.906, -56.916, -119.049]
  MoveL 192 to (6.63, -71.02, 79.57) mm, rotated rx -174.98 ry 26.32 rz -117.81 deg; joints [-15.471, 1.583, -18.407, 73.817, -56.696, -119.04]
  MoveL 193 to (7.97, -72.41, 79.13) mm, rotated rx -175.18 ry 27.05 rz -117.38 deg; joints [-15.496, 1.704, -18.238, 72.683, -56.704, -117.948]
  MoveL 194 to (8.34, -73.51, 79.04) mm, rotated rx -174.99 ry 27.66 rz -117.27 deg; joints [-15.528, 1.7, -18.115, 72.031, -56.302, -117.435]
  MoveL 195 to (8.5, -74.86, 78.73) mm, rotated rx -174.73 ry 28.52 rz -117.1 deg; joints [-15.588, 1.674, -17.952, 71.101, -55.743, -116.691]
  MoveL 196 to (8.44, -76.15, 78.49) mm, rotated rx -172.72 ry 30.25 rz -114.43 deg; joints [-15.723, 1.552, -17.704, 69.121, -54.238, -113.181]
  MoveL 197 to (8.5, -77.42, 78.01) mm, rotated rx -172.45 ry 31.1 rz -114.33 deg; joints [-15.798, 1.526, -17.548, 68.152, -53.692, -112.484]
  MoveL 198 to (8.57, -78.66, 77.54) mm, rotated rx -172.17 ry 31.93 rz -114.22 deg; joints [-15.871, 1.503, -17.397, 67.191, -53.168, -111.784]
  MoveL 199 to (8.69, -79.8, 77.16) mm, rotated rx -171.9 ry 32.67 rz -114.12 deg; joints [-15.935, 1.485, -17.262, 66.331, -52.694, -111.155]
  MoveL 200 to (8.83, -80.8, 76.93) mm, rotated rx -171.63 ry 33.29 rz -114.05 deg; joints [-15.986, 1.466, -17.149, 65.628, -52.254, -110.65]
  MoveL 201 to (8.86, -81.65, 76.86) mm, rotated rx -171.3 ry 33.79 rz -114.04 deg; joints [-16.027, 1.43, -17.059, 65.109, -51.784, -110.308]
  MoveL 202 to (8.62, -82.36, 76.99) mm, rotated rx -170.87 ry 34.19 rz -114.1 deg; joints [-16.061, 1.358, -16.994, 64.807, -51.211, -110.171]
  MoveL 203 to (8.14, -82.88, 77.34) mm, rotated rx -170.34 ry 34.46 rz -114.26 deg; joints [-16.085, 1.251, -16.958, 64.762, -50.545, -110.274]
  MoveL 204 to (8.9, -83.1, 77.88) mm, rotated rx -170.25 ry 34.37 rz -114.24 deg; joints [-16.042, 1.287, -16.962, 64.907, -50.532, -110.36]
  MoveL 205 to (8.4, -83.82, 77.16) mm, rotated rx -175.28 ry 32.13 rz -121.77 deg; joints [-15.881, 1.436, -17.144, 68.063, -52.662, -118.495]
  MoveL 206 to (9.59, -85.18, 76.37) mm, rotated rx -175.55 ry 32.92 rz -121.64 deg; joints [-15.938, 1.548, -16.98, 66.869, -52.596, -117.583]
  MoveL 207 to (10.68, -85.68, 76.53) mm, rotated rx -175.58 ry 33.05 rz -121.63 deg; joints [-15.918, 1.623, -16.944, 66.673, -52.606, -117.444]
  MoveL 208 to (11.92, -86.02, 76.84) mm, rotated rx -175.64 ry 33.03 rz -121.6 deg; joints [-15.879, 1.713, -16.933, 66.641, -52.715, -117.413]
  MoveL 209 to (13.25, -86.21, 77.3) mm, rotated rx -175.67 ry 32.9 rz -121.53 deg; joints [-15.826, 1.808, -16.941, 66.743, -52.87, -117.438]
  MoveL 210 to (11.52, -88.17, 75.33) mm, rotated rx 176.1 ry 27.3 rz -134.76 deg; joints [-15.594, 2.135, -17.19, 71.435, -57.463, -131.842]
  MoveL 211 to (13.08, -89.68, 74.39) mm, rotated rx 175.47 ry 27.94 rz -135.1 deg; joints [-15.647, 2.276, -17.02, 70.374, -57.388, -131.374]
  MoveL 212 to (7.41, -92.83, 71.24) mm, rotated rx 165.08 ry 13.62 rz -156.31 deg; joints [-15.35, 3.01, -17.298, 75.065, -67.641, -155.935]
  MoveL 213 to (6.99, -94.6, 69.39) mm, rotated rx 164.16 ry 14.8 rz -156.93 deg; joints [-15.51, 2.946, -17.033, 73.655, -66.695, -155.359]
  MoveL 214 to (7.01, -96.01, 67.92) mm, rotated rx 163.42 ry 15.71 rz -157.39 deg; joints [-15.633, 2.926, -16.826, 72.509, -66.001, -154.847]
  MoveL 215 to (3.4, -97.81, 66.12) mm, rotated rx 160.45 ry 9.41 rz -165.6 deg; joints [-15.646, 3.148, -16.736, 72.608, -69.699, -164.384]
  MoveL 216 to (4.11, -98.25, 65.89) mm, rotated rx 160.26 ry 9.64 rz -165.75 deg; joints [-15.66, 3.182, -16.686, 72.348, -69.482, -164.301]
  MoveL 217 to (4.55, -99.05, 65.14) mm, rotated rx 159.81 ry 10.1 rz -166 deg; joints [-15.718, 3.197, -16.575, 71.749, -69.084, -164.047]
  MoveL 218 to (1.71, -100.01, 64.3) mm, rotated rx 158.4 ry 4.84 rz -172 deg; joints [-15.716, 3.361, -16.523, 71.702, -71.957, -171.421]
  MoveL 219 to (2.18, -100.59, 63.71) mm, rotated rx 158.03 ry 5.18 rz -172.25 deg; joints [-15.76, 3.374, -16.441, 71.262, -71.59, -171.288]
  MoveL 220 to (2.6, -101.12, 63.22) mm, rotated rx 157.72 ry 5.53 rz -172.5 deg; joints [-15.799, 3.378, -16.368, 70.876, -71.207, -171.191]
  MoveL 221 to (0.07, -101.65, 62.81) mm, rotated rx 157.12 ry 1.3 rz -177.28 deg; joints [-15.802, 3.467, -16.33, 70.757, -73.31, -177.153]
  MoveL 222 to (0.46, -101.9, 62.5) mm, rotated rx 156.93 ry 1.57 rz -177.53 deg; joints [-15.827, 3.465, -16.29, 70.542, -72.966, -177.17]
  MoveL 223 to (0.93, -102.06, 62.36) mm, rotated rx 156.83 ry 1.8 rz -177.76 deg; joints [-15.838, 3.467, -16.268, 70.431, -72.668, -177.226]
  MoveL 224 to (-1.4, -102.13, 62.39) mm, rotated rx 156.83 ry -2.02 rz 177.98 deg; joints [-15.824, 3.527, -16.27, 70.42, -74.51, -182.652]
  MoveL 225 to (-0.93, -102.06, 62.36) mm, rotated rx 156.83 ry -1.8 rz 177.76 deg; joints [-15.826, 3.525, -16.275, 70.43, -74.216, -182.774]
  MoveL 226 to (-0.46, -101.91, 62.5) mm, rotated rx 156.93 ry -1.57 rz 177.54 deg; joints [-15.816, 3.516, -16.296, 70.541, -73.922, -182.94]
  MoveL 227 to (-3.14, -101.52, 62.94) mm, rotated rx 157.51 ry -5.82 rz 172.72 deg; joints [-15.783, 3.572, -16.337, 70.604, -76.011, -189.083]
  MoveL 228 to (-2.61, -101.12, 63.22) mm, rotated rx 157.72 ry -5.53 rz 172.5 deg; joints [-15.762, 3.559, -16.388, 70.854, -75.702, -189.295]
  MoveL 229 to (-2.18, -100.59, 63.71) mm, rotated rx 158.03 ry -5.18 rz 172.24 deg; joints [-15.729, 3.524, -16.458, 71.232, -75.342, -189.573]
  MoveL 230 to (-5.22, -99.67, 64.64) mm, rotated rx 159.48 ry -10.41 rz 166.17 deg; joints [-15.671, 3.63, -16.54, 71.222, -78.128, -197.168]
  MoveL 231 to (-4.55, -99.05, 65.14) mm, rotated rx 159.81 ry -10.1 rz 166 deg; joints [-15.63, 3.626, -16.624, 71.633, -77.889, -197.393]
  MoveL 232 to (-4.11, -98.25, 65.89) mm, rotated rx 160.27 ry -9.64 rz 165.75 deg; joints [-15.578, 3.582, -16.731, 72.2, -77.538, -197.711]
  MoveL 233 to (-7.39, -97.12, 66.82) mm, rotated rx 162.82 ry -16.38 rz 157.71 deg; joints [-15.54, 3.829, -16.77, 71.378, -81.442, -207.181]
  MoveL 234 to (-7.01, -96.01, 67.92) mm, rotated rx 163.42 ry -15.72 rz 157.38 deg; joints [-15.463, 3.763, -16.921, 72.174, -81.052, -207.577]
  MoveL 235 to (-7, -94.6, 69.39) mm, rotated rx 164.17 ry -14.81 rz 156.92 deg; joints [-15.371, 3.636, -17.112, 73.215, -80.491, -208.129]
  MoveL 236 to (-7.48, -92.8, 71.26) mm, rotated rx 165.15 ry -13.79 rz 156.11 deg; joints [-15.262, 3.451, -17.348, 74.505, -79.854, -209.094]
  MoveL 237 to (-13.13, -89.63, 74.43) mm, rotated rx 175.61 ry -28.07 rz 134.85 deg; joints [-15.239, 4.306, -17.25, 69.785, -89.701, -230.616]
  MoveL 238 to (-11.56, -88.14, 75.37) mm, rotated rx 176.25 ry -27.43 rz 134.5 deg; joints [-15.148, 4.371, -17.444, 70.572, -89.67, -231.094]
  MoveL 239 to (-13.24, -86.21, 77.29) mm, rotated rx -175.7 ry -32.89 rz 121.58 deg; joints [-15.214, 4.82, -17.286, 66.859, -93.953, -242.196]
  MoveL 240 to (-11.92, -86.02, 76.84) mm, rotated rx -175.64 ry -33.03 rz 121.6 deg; joints [-15.224, 4.938, -17.301, 66.771, -94.063, -242.181]
  MoveL 241 to (-10.68, -85.68, 76.53) mm, rotated rx -175.58 ry -33.05 rz 121.63 deg; joints [-15.223, 5.038, -17.334, 66.788, -94.12, -242.188]
  MoveL 242 to (-9.59, -85.18, 76.37) mm, rotated rx -175.55 ry -32.92 rz 121.64 deg; joints [-15.212, 5.11, -17.387, 66.917, -94.088, -242.228]
  MoveL 243 to (-8.43, -83.79, 77.19) mm, rotated rx -175.04 ry -32.26 rz 121.39 deg; joints [-15.132, 5.162, -17.564, 67.623, -94.128, -242.634]
  MoveL 244 to (-8.89, -83.12, 77.86) mm, rotated rx -170.36 ry -34.33 rz 114.4 deg; joints [-15.2, 5.396, -17.434, 65.454, -96.038, -248.222]
  MoveL 245 to (-8.17, -82.86, 77.3) mm, rotated rx -170.42 ry -34.43 rz 114.32 deg; joints [-15.224, 5.452, -17.438, 65.321, -95.958, -248.272]
  MoveL 246 to (-8.66, -82.3, 76.95) mm, rotated rx -170.97 ry -34.14 rz 114.17 deg; joints [-15.244, 5.337, -17.453, 65.339, -95.242, -248.451]
  MoveL 247 to (-8.87, -81.54, 76.84) mm, rotated rx -171.41 ry -33.7 rz 114.11 deg; joints [-15.242, 5.245, -17.508, 65.555, -94.631, -248.594]
  MoveL 248 to (-8.81, -80.61, 76.95) mm, rotated rx -171.74 ry -33.15 rz 114.14 deg; joints [-15.22, 5.176, -17.596, 65.942, -94.124, -248.708]
  MoveL 249 to (-8.67, -79.52, 77.23) mm, rotated rx -172.02 ry -32.47 rz 114.23 deg; joints [-15.183, 5.108, -17.712, 66.479, -93.638, -248.817]
  MoveL 250 to (-8.55, -78.28, 77.67) mm, rotated rx -172.31 ry -31.65 rz 114.34 deg; joints [-15.134, 5.029, -17.851, 67.141, -93.121, -248.938]
  MoveL 251 to (-8.49, -76.94, 78.18) mm, rotated rx -172.6 ry -30.75 rz 114.46 deg; joints [-15.081, 4.938, -18.004, 67.878, -92.57, -249.079]
  MoveL 252 to (-8.51, -75.85, 78.43) mm, rotated rx -174.61 ry -29.14 rz 117.08 deg; joints [-15.019, 4.733, -18.19, 69.315, -91.216, -247.146]
  MoveL 253 to (-8.47, -74.37, 78.86) mm, rotated rx -174.92 ry -28.15 rz 117.29 deg; joints [-14.972, 4.635, -18.36, 70.138, -90.615, -247.217]
  MoveL 254 to (-8.24, -73.1, 79.09) mm, rotated rx -175.16 ry -27.37 rz 117.44 deg; joints [-14.939, 4.574, -18.501, 70.788, -90.141, -247.29]
  MoveL 255 to (-7.81, -72.09, 79.1) mm, rotated rx -175.33 ry -26.84 rz 117.53 deg; joints [-14.922, 4.553, -18.608, 71.229, -89.799, -247.36]
  MoveL 256 to (-6.43, -70.76, 79.48) mm, rotated rx -175.11 ry -26.17 rz 117.96 deg; joints [-14.863, 4.638, -18.793, 72.015, -89.896, -247.231]
  MoveL 257 to (-7.32, -70.96, 78.29) mm, rotated rx -175.84 ry -26.46 rz 117.3 deg; joints [-14.957, 4.51, -18.675, 71.344, -89.033, -247.65]
  MoveL 258 to (-7.42, -70.56, 77.72) mm, rotated rx -176.24 ry -26.35 rz 117.05 deg; joints [-14.993, 4.451, -18.675, 71.246, -88.491, -247.87]
  MoveL 259 to (-6.7, -70.14, 77.26) mm, rotated rx -177.88 ry -25.39 rz 119.51 deg; joints [-14.989, 4.376, -18.762, 72.008, -87.526, -245.814]
  MoveL 260 to (-5.92, -69.96, 76.53) mm, rotated rx -177.91 ry -25.64 rz 119.37 deg; joints [-15.024, 4.453, -18.75, 71.754, -87.526, -245.898]
  MoveL 261 to (-5.02, -69.82, 75.79) mm, rotated rx -177.88 ry -25.94 rz 119.25 deg; joints [-15.058, 4.549, -18.737, 71.479, -87.597, -245.964]
  MoveL 262 to (-3.99, -69.56, 75.15) mm, rotated rx -177.8 ry -26.15 rz 119.21 deg; joints [-15.082, 4.654, -18.745, 71.312, -87.717, -245.987]
  MoveL 263 to (-2.94, -69.02, 74.77) mm, rotated rx -177.71 ry -26.12 rz 119.3 deg; joints [-15.086, 4.746, -18.799, 71.398, -87.801, -245.959]
  MoveL 264 to (-2.49, -68.6, 74.25) mm, rotated rx -177.85 ry -26.1 rz 119.19 deg; joints [-15.11, 4.765, -18.817, 71.348, -87.59, -246.065]
  MoveL 265 to (-2.05, -68.18, 73.73) mm, rotated rx -178.01 ry -26.07 rz 119.08 deg; joints [-15.134, 4.782, -18.835, 71.298, -87.37, -246.174]
  MoveL 266 to (-1.64, -67.79, 73.2) mm, rotated rx -178.2 ry -26.04 rz 119 deg; joints [-15.159, 4.794, -18.85, 71.241, -87.124, -246.251]
  Set speed (50.0 mm/s)
  MoveL 267 to (-1.64, -67.79, 73.2) mm, rotated rx -178.2 ry -26.04 rz 119 deg; joints [-15.159, 4.794, -18.85, 71.241, -87.124, -246.251]
  MoveL 268 to (-3.35, -139.46, 142.95) mm, rotated rx 165.22 ry -11.47 rz 146.16 deg; joints [-11.389, 2.134, -14.376, 73.889, -79.145, -216.161]
  Set speed (50.0 mm/s)
  MoveL 269 to (3.35, -139.46, 142.95) mm, rotated rx 164.3 ry -10.15 rz 144.74 deg; joints [-11.355, 2.358, -14.405, 73.913, -77.143, -217.209]
  MoveL 270 to (3.35, -68.75, 72.24) mm, rotated rx 164.3 ry -10.15 rz 144.74 deg; joints [-15.25, 3.252, -18.966, 75.969, -72.353, -220.766]
  MoveL 271 to (1.63, -67.79, 73.2) mm, rotated rx 155.51 ry 9.41 rz 166.61 deg; joints [-15.798, 1.644, -18.484, 72.688, -58.86, -191.342]
  Set speed (10.0 mm/s)
  MoveL 272 to (2.07, -68.2, 73.76) mm, rotated rx 155.54 ry 9.56 rz 166.4 deg; joints [-15.768, 1.64, -18.47, 72.794, -58.687, -191.517]
  MoveL 273 to (2.53, -68.64, 74.3) mm, rotated rx 155.55 ry 9.71 rz 166.22 deg; joints [-15.738, 1.639, -18.452, 72.873, -58.521, -191.663]
  MoveL 274 to (3.06, -69.11, 74.82) mm, rotated rx 155.54 ry 9.84 rz 166.07 deg; joints [-15.708, 1.647, -18.431, 72.918, -58.387, -191.764]
  MoveL 275 to (4.19, -69.63, 75.26) mm, rotated rx 155.53 ry 9.74 rz 166.19 deg; joints [-15.663, 1.734, -18.403, 72.823, -58.562, -191.637]
  MoveL 276 to (5.25, -69.87, 75.97) mm, rotated rx 155.76 ry 9.61 rz 166.19 deg; joints [-15.595, 1.808, -18.422, 73.065, -58.781, -191.856]
  MoveL 277 to (6.16, -70.02, 76.76) mm, rotated rx 156.06 ry 9.52 rz 166.11 deg; joints [-15.526, 1.864, -18.454, 73.413, -58.948, -192.203]
  MoveL 278 to (6.84, -70.15, 77.58) mm, rotated rx 155.78 ry 11.18 rz 167.75 deg; joints [-15.529, 1.8, -18.399, 72.916, -58.015, -189.751]
  MoveL 279 to (7.69, -70.84, 77.79) mm, rotated rx 155.56 ry 11.25 rz 167.76 deg; joints [-15.514, 1.85, -18.34, 72.636, -57.944, -189.518]
  MoveL 280 to (6.15, -70.44, 79.2) mm, rotated rx 156.14 ry 12.03 rz 166.57 deg; joints [-15.485, 1.581, -18.448, 73.906, -56.916, -191.049]
  MoveL 281 to (6.63, -71.02, 79.57) mm, rotated rx 156.01 ry 12.22 rz 166.41 deg; joints [-15.471, 1.583, -18.407, 73.817, -56.696, -191.04]
  MoveL 282 to (7.97, -72.41, 79.13) mm, rotated rx 155.24 ry 12.22 rz 166.77 deg; joints [-15.496, 1.704, -18.238, 72.683, -56.704, -189.948]
  MoveL 283 to (8.34, -73.51, 79.04) mm, rotated rx 154.67 ry 12.53 rz 166.67 deg; joints [-15.528, 1.7, -18.115, 72.031, -56.302, -189.435]
  MoveL 284 to (8.5, -74.86, 78.73) mm, rotated rx 153.87 ry 12.96 rz 166.54 deg; joints [-15.588, 1.674, -17.952, 71.101, -55.743, -188.691]
  MoveL 285 to (8.44, -76.15, 78.49) mm, rotated rx 152.54 ry 15.06 rz 167.9 deg; joints [-15.723, 1.552, -17.704, 69.121, -54.238, -185.181]
  MoveL 286 to (8.5, -77.42, 78.01) mm, rotated rx 151.73 ry 15.47 rz 167.64 deg; joints [-15.798, 1.526, -17.548, 68.152, -53.692, -184.484]
  MoveL 287 to (8.57, -78.66, 77.54) mm, rotated rx 150.93 ry 15.87 rz 167.39 deg; joints [-15.871, 1.503, -17.397, 67.191, -53.168, -183.784]
  MoveL 288 to (8.69, -79.8, 77.16) mm, rotated rx 150.23 ry 16.24 rz 167.16 deg; joints [-15.935, 1.485, -17.262, 66.331, -52.694, -183.155]
  MoveL 289 to (8.83, -80.8, 76.93) mm, rotated rx 149.64 ry 16.58 rz 166.91 deg; joints [-15.986, 1.466, -17.149, 65.628, -52.254, -182.65]
  MoveL 290 to (8.86, -81.65, 76.86) mm, rotated rx 149.18 ry 16.94 rz 166.61 deg; joints [-16.027, 1.43, -17.059, 65.109, -51.784, -182.308]
  MoveL 291 to (8.62, -82.36, 76.99) mm, rotated rx 148.84 ry 17.36 rz 166.21 deg; joints [-16.061, 1.358, -16.994, 64.807, -51.211, -182.171]
  MoveL 292 to (8.14, -82.88, 77.34) mm, rotated rx 148.64 ry 17.84 rz 165.7 deg; joints [-16.085, 1.251, -16.958, 64.762, -50.545, -182.274]
  MoveL 293 to (8.9, -83.1, 77.88) mm, rotated rx 148.75 ry 17.9 rz 165.7 deg; joints [-16.042, 1.287, -16.962, 64.907, -50.532, -182.36]
  MoveL 294 to (8.4, -83.82, 77.16) mm, rotated rx 150.15 ry 13.33 rz 161.31 deg; joints [-15.881, 1.436, -17.144, 68.063, -52.662, -190.495]
  MoveL 295 to (9.59, -85.18, 76.37) mm, rotated rx 149.31 ry 13.29 rz 161.38 deg; joints [-15.938, 1.548, -16.98, 66.869, -52.596, -189.583]
  MoveL 296 to (10.68, -85.68, 76.53) mm, rotated rx 149.18 ry 13.29 rz 161.38 deg; joints [-15.918, 1.623, -16.944, 66.673, -52.606, -189.444]
  MoveL 297 to (11.92, -86.02, 76.84) mm, rotated rx 149.18 ry 13.24 rz 161.44 deg; joints [-15.879, 1.713, -16.933, 66.641, -52.715, -189.413]
  MoveL 298 to (13.25, -86.21, 77.3) mm, rotated rx 149.3 ry 13.19 rz 161.55 deg; joints [-15.826, 1.808, -16.941, 66.743, -52.87, -189.438]
  MoveL 299 to (11.52, -88.17, 75.33) mm, rotated rx 152.84 ry 4.84 rz 153.02 deg; joints [-15.594, 2.135, -17.19, 71.435, -57.463, -203.842]
  MoveL 300 to (13.08, -89.68, 74.39) mm, rotated rx 152.05 ry 4.49 rz 152.91 deg; joints [-15.647, 2.276, -17.02, 70.374, -57.388, -203.374]
  MoveL 301 to (7.41, -92.83, 71.24) mm, rotated rx 162.21 ry -9.51 rz 134.98 deg; joints [-15.35, 3.01, -17.298, 75.065, -67.641, -227.935]
  MoveL 302 to (6.99, -94.6, 69.39) mm, rotated rx 160.76 ry -9.9 rz 134.83 deg; joints [-15.51, 2.946, -17.033, 73.655, -66.695, -227.359]
  MoveL 303 to (8.15, -92.88, 72.03) mm, rotated rx 162.05 ry -8.99 rz 134.45 deg; joints [-15.312, 2.967, -17.327, 75.425, -67.041, -228.448]
  MoveL 304 to (5.46, -94.88, 70.13) mm, rotated rx 166.92 ry -13.95 rz 125.95 deg; joints [-15.315, 3.305, -17.223, 75.247, -71.125, -237.643]
  MoveL 305 to (6.15, -95.3, 69.93) mm, rotated rx 166.63 ry -14.02 rz 125.9 deg; joints [-15.326, 3.336, -17.175, 75.017, -70.905, -237.592]
  MoveL 306 to (6.57, -96.1, 69.26) mm, rotated rx 166.05 ry -14.25 rz 125.85 deg; joints [-15.377, 3.345, -17.067, 74.465, -70.5, -237.391]
  MoveL 307 to (4.46, -97.28, 68.24) mm, rotated rx 170.49 ry -17.38 rz 118.96 deg; joints [-15.378, 3.596, -16.994, 74.171, -73.585, -244.363]
  MoveL 308 to (4.91, -97.85, 67.7) mm, rotated rx 170.03 ry -17.58 rz 118.88 deg; joints [-15.417, 3.605, -16.913, 73.764, -73.216, -244.272]
  MoveL 309 to (5.31, -98.38, 67.24) mm, rotated rx 169.58 ry -17.74 rz 118.77 deg; joints [-15.452, 3.605, -16.84, 73.403, -72.827, -244.213]
  MoveL 310 to (3.37, -99.13, 66.62) mm, rotated rx 173.35 ry -19.71 rz 113 deg; joints [-15.463, 3.758, -16.779, 73.077, -75.039, -249.765]
  MoveL 311 to (3.74, -99.39, 66.32) mm, rotated rx 173.01 ry -19.79 rz 112.86 deg; joints [-15.486, 3.753, -16.739, 72.875, -74.691, -249.808]
  MoveL 312 to (0.93, -102.06, 62.36) mm, rotated rx 170.65 ry -21.36 rz 112.38 deg; joints [-15.838, 3.467, -16.268, 70.431, -72.668, -249.226]
  MoveL 313 to (-1.4, -102.13, 62.39) mm, rotated rx 174.53 ry -22.63 rz 106.66 deg; joints [-15.824, 3.527, -16.27, 70.42, -74.51, -254.652]
  MoveL 314 to (-0.93, -102.06, 62.36) mm, rotated rx 174.3 ry -22.56 rz 106.53 deg; joints [-15.826, 3.525, -16.275, 70.43, -74.216, -254.774]
  MoveL 315 to (-0.46, -101.91, 62.5) mm, rotated rx 174.1 ry -22.4 rz 106.39 deg; joints [-15.816, 3.516, -16.296, 70.541, -73.922, -254.94]
  MoveL 316 to (-3.14, -101.52, 62.94) mm, rotated rx 178.68 ry -23.15 rz 99.84 deg; joints [-15.783, 3.572, -16.337, 70.604, -76.011, -261.083]
  MoveL 317 to (-2.61, -101.12, 63.22) mm, rotated rx 178.45 ry -22.88 rz 99.72 deg; joints [-15.762, 3.559, -16.388, 70.854, -75.702, -261.295]
  MoveL 318 to (-2.18, -100.59, 63.71) mm, rotated rx 178.19 ry -22.47 rz 99.6 deg; joints [-15.729, 3.524, -16.458, 71.232, -75.342, -261.573]
  MoveL 319 to (-5.22, -99.67, 64.64) mm, rotated rx -175.94 ry -22.57 rz 91.47 deg; joints [-15.671, 3.63, -16.54, 71.222, -78.128, -269.168]
  MoveL 320 to (-4.55, -99.05, 65.14) mm, rotated rx -176.18 ry -22.17 rz 91.45 deg; joints [-15.63, 3.626, -16.624, 71.633, -77.889, -269.394]
  MoveL 321 to (-4.11, -98.25, 65.89) mm, rotated rx -176.52 ry -21.61 rz 91.4 deg; joints [-15.578, 3.582, -16.731, 72.2, -77.538, -269.711]
  MoveL 322 to (-7.39, -97.12, 66.82) mm, rotated rx -168.85 ry -20.89 rz 81.15 deg; joints [-15.54, 3.829, -16.77, 71.378, -81.442, -279.181]
  MoveL 323 to (-7.01, -96.01, 67.92) mm, rotated rx -169.39 ry -20.18 rz 81.18 deg; joints [-15.463, 3.763, -16.921, 72.174, -81.052, -279.577]
  MoveL 324 to (-7, -94.6, 69.39) mm, rotated rx -170.14 ry -19.26 rz 81.17 deg; joints [-15.371, 3.636, -17.112, 73.215, -80.491, -280.129]
  MoveL 325 to (-7.48, -92.8, 71.26) mm, rotated rx -170.93 ry -18.08 rz 80.86 deg; joints [-15.262, 3.451, -17.348, 74.505, -79.854, -281.094]
  MoveL 326 to (-13.13, -89.63, 74.43) mm, rotated rx -154.13 ry -12.1 rz 58.96 deg; joints [-15.239, 4.306, -17.25, 69.785, -89.701, -302.616]
  MoveL 327 to (-11.56, -88.14, 75.37) mm, rotated rx -154.62 ry -11.39 rz 59.01 deg; joints [-15.148, 4.371, -17.444, 70.572, -89.67, -303.094]
  MoveL 328 to (-13.24, -86.21, 77.29) mm, rotated rx -147.38 ry -6.19 rz 49.04 deg; joints [-15.214, 4.82, -17.286, 66.859, -93.953, -314.196]
  MoveL 329 to (-11.92, -86.02, 76.84) mm, rotated rx -147.23 ry -6.19 rz 49.07 deg; joints [-15.224, 4.938, -17.301, 66.771, -94.063, -314.181]
  MoveL 330 to (-10.68, -85.68, 76.53) mm, rotated rx -147.2 ry -6.15 rz 49.13 deg; joints [-15.223, 5.038, -17.334, 66.788, -94.12, -314.188]
  MoveL 331 to (-9.59, -85.18, 76.37) mm, rotated rx -147.32 ry -6.08 rz 49.17 deg; joints [-15.212, 5.11, -17.387, 66.917, -94.088, -314.228]
  MoveL 332 to (-8.43, -83.79, 77.2) mm, rotated rx -147.82 ry -5.47 rz 49.25 deg; joints [-15.132, 5.162, -17.564, 67.623, -94.128, -314.634]
  MoveL 333 to (-8.89, -83.11, 77.87) mm, rotated rx -144.54 ry -2.41 rz 44.55 deg; joints [-15.201, 5.399, -17.433, 65.428, -96.059, -320.286]
  MoveL 334 to (-8.21, -82.82, 77.28) mm, rotated rx -144.5 ry -2.53 rz 44.39 deg; joints [-15.227, 5.445, -17.437, 65.291, -95.919, -320.351]
  MoveL 335 to (-8.72, -82.18, 76.93) mm, rotated rx -144.98 ry -2.87 rz 43.93 deg; joints [-15.246, 5.323, -17.458, 65.338, -95.155, -320.54]
  MoveL 336 to (-8.87, -81.32, 76.87) mm, rotated rx -145.57 ry -3.05 rz 43.68 deg; joints [-15.238, 5.23, -17.525, 65.61, -94.524, -320.687]
  MoveL 337 to (-8.76, -80.28, 77.04) mm, rotated rx -146.26 ry -3.1 rz 43.58 deg; joints [-15.209, 5.158, -17.629, 66.073, -93.992, -320.808]
  MoveL 338 to (-8.6, -79.04, 77.41) mm, rotated rx -147.09 ry -3.08 rz 43.57 deg; joints [-15.165, 5.082, -17.763, 66.7, -93.46, -320.932]
  MoveL 339 to (-8.51, -77.65, 77.92) mm, rotated rx -148.04 ry -3.02 rz 43.57 deg; joints [-15.11, 4.991, -17.919, 67.45, -92.886, -321.075]
  MoveL 340 to (-8.5, -76.45, 78.23) mm, rotated rx -150.19 ry -4.12 rz 45.28 deg; joints [-15.04, 4.782, -18.119, 68.944, -91.513, -319.196]
  MoveL 341 to (-8.51, -75.06, 78.67) mm, rotated rx -151.17 ry -4.08 rz 45.41 deg; joints [-14.994, 4.685, -18.278, 69.726, -90.939, -319.26]
  MoveL 342 to (-8.4, -73.8, 78.99) mm, rotated rx -152.01 ry -4.03 rz 45.51 deg; joints [-14.957, 4.611, -18.421, 70.404, -90.449, -319.329]
  MoveL 343 to (-8.12, -72.75, 79.12) mm, rotated rx -152.65 ry -3.99 rz 45.58 deg; joints [-14.932, 4.571, -18.537, 70.92, -90.069, -319.397]
  MoveL 344 to (-7.69, -71.91, 79.08) mm, rotated rx -153.09 ry -3.98 rz 45.62 deg; joints [-14.921, 4.56, -18.625, 71.267, -89.787, -319.462]
  MoveL 345 to (-6.35, -70.68, 79.46) mm, rotated rx -153.61 ry -3.59 rz 46.16 deg; joints [-14.864, 4.647, -18.798, 72.001, -89.922, -319.33]
  MoveL 346 to (-7.32, -70.96, 78.3) mm, rotated rx -153.52 ry -4.3 rz 45.18 deg; joints [-14.958, 4.515, -18.673, 71.311, -89.072, -319.74]
  MoveL 347 to (-7.5, -70.64, 77.74) mm, rotated rx -153.71 ry -4.62 rz 44.75 deg; joints [-14.994, 4.452, -18.664, 71.185, -88.535, -319.959]
  MoveL 348 to (-6.9, -70.26, 77.33) mm, rotated rx -155.12 ry -5.79 rz 46.68 deg; joints [-14.988, 4.362, -18.749, 71.976, -87.533, -317.836]
  MoveL 349 to (-6.06, -69.99, 76.66) mm, rotated rx -154.94 ry -5.85 rz 46.56 deg; joints [-15.018, 4.442, -18.752, 71.792, -87.54, -317.901]
  MoveL 350 to (-5.15, -69.84, 75.89) mm, rotated rx -154.65 ry -5.92 rz 46.41 deg; joints [-15.054, 4.537, -18.738, 71.507, -87.602, -317.972]
  MoveL 351 to (-4.1, -69.6, 75.21) mm, rotated rx -154.4 ry -5.93 rz 46.35 deg; joints [-15.08, 4.645, -18.742, 71.315, -87.72, -318.002]
  MoveL 352 to (-2.99, -69.06, 74.8) mm, rotated rx -154.38 ry -5.84 rz 46.49 deg; joints [-15.085, 4.744, -18.795, 71.39, -87.825, -317.972]
  MoveL 353 to (-2.52, -68.62, 74.28) mm, rotated rx -154.45 ry -5.95 rz 46.33 deg; joints [-15.108, 4.765, -18.816, 71.346, -87.613, -318.077]
  MoveL 354 to (-2.07, -68.19, 73.75) mm, rotated rx -154.52 ry -6.07 rz 46.15 deg; joints [-15.133, 4.783, -18.835, 71.295, -87.386, -318.189]
  MoveL 355 to (-1.64, -67.79, 73.2) mm, rotated rx -154.6 ry -6.23 rz 45.99 deg; joints [-15.159, 4.796, -18.85, 71.236, -87.132, -318.269]
  Set speed (50.0 mm/s)
  MoveL 356 to (-1.64, -67.79, 73.2) mm, rotated rx -154.6 ry -6.23 rz 45.99 deg; joints [-15.159, 4.796, -18.85, 71.236, -87.132, -318.269]
  MoveL 357 to (-3.35, -139.46, 142.95) mm, rotated rx -173.27 ry -17.41 rz 71.64 deg; joints [-11.389, 2.134, -14.376, 73.889, -79.145, -288.161]
  Set speed (50.0 mm/s)
  MoveL 358 to (3.35, -139.46, 142.95) mm, rotated rx -174.85 ry -17.93 rz 70.52 deg; joints [-11.355, 2.358, -14.405, 73.913, -77.143, -289.209]
  MoveL 359 to (3.35, -68.75, 72.24) mm, rotated rx -174.85 ry -17.93 rz 70.52 deg; joints [-15.25, 3.252, -18.966, 75.969, -72.353, -292.766]
  MoveL 360 to (1.63, -67.79, 73.2) mm, rotated rx 162.57 ry -19.78 rz 99.72 deg; joints [-15.798, 1.644, -18.484, 72.688, -58.86, -263.342]
  Set speed (10.0 mm/s)
  MoveL 361 to (2.07, -68.2, 73.76) mm, rotated rx 162.43 ry -19.69 rz 99.56 deg; joints [-15.768, 1.64, -18.47, 72.794, -58.687, -263.517]
  MoveL 362 to (2.53, -68.64, 74.3) mm, rotated rx 162.29 ry -19.63 rz 99.41 deg; joints [-15.738, 1.639, -18.452, 72.873, -58.521, -263.663]
  MoveL 363 to (3.06, -69.11, 74.82) mm, rotated rx 162.17 ry -19.59 rz 99.31 deg; joints [-15.708, 1.647, -18.431, 72.918, -58.387, -263.764]
  MoveL 364 to (4.19, -69.63, 75.26) mm, rotated rx 162.25 ry -19.64 rz 99.41 deg; joints [-15.663, 1.734, -18.403, 72.823, -58.563, -263.637]
  MoveL 365 to (5.25, -69.87, 75.97) mm, rotated rx 162.47 ry -19.47 rz 99.29 deg; joints [-15.595, 1.808, -18.422, 73.065, -58.781, -263.856]
  MoveL 366 to (6.16, -70.02, 76.76) mm, rotated rx 162.68 ry -19.24 rz 99.09 deg; joints [-15.526, 1.864, -18.454, 73.413, -58.948, -264.204]
  MoveL 367 to (6.84, -70.15, 77.58) mm, rotated rx 160.96 ry -18.84 rz 101.34 deg; joints [-15.529, 1.8, -18.399, 72.916, -58.015, -261.751]
  MoveL 368 to (7.69, -70.84, 77.79) mm, rotated rx 160.8 ry -19 rz 101.45 deg; joints [-15.514, 1.85, -18.34, 72.636, -57.944, -261.518]
  MoveL 369 to (6.15, -70.44, 79.2) mm, rotated rx 160.28 ry -18.17 rz 100.3 deg; joints [-15.485, 1.581, -18.448, 73.906, -56.916, -263.049]
  MoveL 370 to (6.63, -71.02, 79.57) mm, rotated rx 160.05 ry -18.21 rz 100.24 deg; joints [-15.471, 1.583, -18.407, 73.817, -56.696, -263.04]
  MoveL 371 to (7.97, -72.41, 79.13) mm, rotated rx 159.72 ry -18.9 rz 100.87 deg; joints [-15.496, 1.704, -18.238, 72.683, -56.704, -261.948]
  MoveL 372 to (8.34, -73.51, 79.04) mm, rotated rx 159.18 ry -19.28 rz 101.07 deg; joints [-15.528, 1.7, -18.115, 72.031, -56.302, -261.435]
  MoveL 373 to (8.5, -74.86, 78.73) mm, rotated rx 158.43 ry -19.81 rz 101.37 deg; joints [-15.588, 1.674, -17.952, 71.101, -55.743, -260.691]
  MoveL 374 to (8.44, -76.15, 78.49) mm, rotated rx 155.82 ry -20.08 rz 103.94 deg; joints [-15.723, 1.552, -17.704, 69.121, -54.238, -257.181]
  MoveL 375 to (8.5, -77.42, 78.01) mm, rotated rx 155.06 ry -20.6 rz 104.16 deg; joints [-15.798, 1.526, -17.548, 68.152, -53.692, -256.484]
  MoveL 376 to (8.57, -78.66, 77.54) mm, rotated rx 154.31 ry -21.1 rz 104.39 deg; joints [-15.871, 1.503, -17.397, 67.191, -53.168, -255.784]
  MoveL 377 to (8.69, -79.8, 77.16) mm, rotated rx 153.63 ry -21.53 rz 104.6 deg; joints [-15.935, 1.485, -17.262, 66.331, -52.694, -255.155]
  MoveL 378 to (8.83, -80.8, 76.93) mm, rotated rx 153.02 ry -21.87 rz 104.75 deg; joints [-15.986, 1.466, -17.149, 65.628, -52.254, -254.65]
  MoveL 379 to (8.86, -81.65, 76.86) mm, rotated rx 152.45 ry -22.09 rz 104.8 deg; joints [-16.027, 1.43, -17.059, 65.109, -51.784, -254.308]
  MoveL 380 to (8.62, -82.36, 76.99) mm, rotated rx 151.88 ry -22.18 rz 104.71 deg; joints [-16.061, 1.358, -16.994, 64.807, -51.211, -254.171]
  MoveL 381 to (8.14, -82.88, 77.34) mm, rotated rx 151.33 ry -22.11 rz 104.46 deg; joints [-16.085, 1.251, -16.958, 64.762, -50.545, -254.274]
  MoveL 382 to (8.9, -83.1, 77.88) mm, rotated rx 151.33 ry -21.99 rz 104.43 deg; joints [-16.042, 1.287, -16.962, 64.907, -50.532, -254.36]
  MoveL 383 to (8.4, -83.82, 77.16) mm, rotated rx 156.39 ry -22.91 rz 97.72 deg; joints [-15.881, 1.436, -17.144, 68.063, -52.662, -262.495]
  MoveL 384 to (9.59, -85.18, 76.37) mm, rotated rx 156.03 ry -23.66 rz 98.13 deg; joints [-15.938, 1.548, -16.98, 66.869, -52.596, -261.583]
  MoveL 385 to (10.68, -85.68, 76.53) mm, rotated rx 155.96 ry -23.78 rz 98.19 deg; joints [-15.918, 1.623, -16.944, 66.673, -52.606, -261.444]
  MoveL 386 to (11.92, -86.02, 76.84) mm, rotated rx 156.02 ry -23.8 rz 98.23 deg; joints [-15.879, 1.713, -16.933, 66.641, -52.715, -261.413]
  MoveL 387 to (13.25, -86.21, 77.3) mm, rotated rx 156.12 ry -23.72 rz 98.27 deg; joints [-15.826, 1.808, -16.941, 66.743, -52.87, -261.438]
  MoveL 388 to (11.52, -88.17, 75.33) mm, rotated rx 166.02 ry -23.99 rz 85.18 deg; joints [-15.594, 2.135, -17.19, 71.435, -57.463, -275.842]
  MoveL 389 to (13.08, -89.68, 74.39) mm, rotated rx 166.04 ry -24.84 rz 85.11 deg; joints [-15.647, 2.276, -17.02, 70.374, -57.388, -275.374]
  MoveL 390 to (7.41, -92.83, 71.24) mm, rotated rx -176.1 ry -19.73 rz 60.8 deg; joints [-15.35, 3.01, -17.298, 75.065, -67.641, -299.935]
  MoveL 391 to (6.99, -94.6, 69.39) mm, rotated rx -176.11 ry -21.21 rz 60.42 deg; joints [-15.51, 2.946, -17.033, 73.655, -66.695, -299.359]
  MoveL 392 to (7.01, -96.01, 67.92) mm, rotated rx -176.09 ry -22.37 rz 60.14 deg; joints [-15.633, 2.926, -16.826, 72.509, -66.001, -298.847]
  MoveL 393 to (3.4, -97.81, 66.12) mm, rotated rx -169.58 ry -19.04 rz 50.27 deg; joints [-15.646, 3.148, -16.736, 72.608, -69.699, -308.384]
  MoveL 394 to (4.11, -98.25, 65.89) mm, rotated rx -169.57 ry -19.34 rz 50.15 deg; joints [-15.66, 3.182, -16.686, 72.348, -69.482, -308.301]
  MoveL 395 to (4.55, -99.05, 65.14) mm, rotated rx -169.47 ry -19.97 rz 49.94 deg; joints [-15.718, 3.197, -16.575, 71.749, -69.084, -308.047]
  MoveL 396 to (1.71, -100.01, 64.3) mm, rotated rx -165.06 ry -16.49 rz 42.74 deg; joints [-15.716, 3.361, -16.523, 71.702, -71.957, -315.421]
  MoveL 397 to (2.18, -100.59, 63.71) mm, rotated rx -164.95 ry -16.98 rz 42.5 deg; joints [-15.76, 3.374, -16.441, 71.262, -71.59, -315.288]
  MoveL 398 to (2.6, -101.12, 63.22) mm, rotated rx -164.89 ry -17.45 rz 42.25 deg; joints [-15.799, 3.378, -16.368, 70.876, -71.207, -315.191]
  MoveL 399 to (0.07, -101.65, 62.81) mm, rotated rx -161.89 ry -14.29 rz 36.69 deg; joints [-15.802, 3.467, -16.33, 70.757, -73.31, -321.152]
  MoveL 400 to (0.46, -101.9, 62.5) mm, rotated rx -161.89 ry -14.62 rz 36.44 deg; joints [-15.827, 3.465, -16.29, 70.542, -72.966, -321.17]
  MoveL 401 to (0.93, -102.06, 62.36) mm, rotated rx -161.94 ry -14.86 rz 36.24 deg; joints [-15.838, 3.467, -16.268, 70.431, -72.668, -321.226]
  MoveL 402 to (-1.4, -102.13, 62.39) mm, rotated rx -159.76 ry -11.69 rz 31.47 deg; joints [-15.824, 3.527, -16.27, 70.42, -74.51, -326.652]
  MoveL 403 to (-0.93, -102.06, 62.36) mm, rotated rx -159.88 ry -11.87 rz 31.28 deg; joints [-15.826, 3.525, -16.275, 70.43, -74.216, -326.774]
  MoveL 404 to (-0.46, -101.91, 62.5) mm, rotated rx -160.1 ry -12.01 rz 31.1 deg; joints [-15.816, 3.516, -16.296, 70.541, -73.922, -326.94]
  MoveL 405 to (-3.14, -101.52, 62.94) mm, rotated rx -158.21 ry -8.15 rz 26 deg; joints [-15.783, 3.572, -16.337, 70.604, -76.01, -333.083]
  MoveL 406 to (-2.61, -101.12, 63.22) mm, rotated rx -158.54 ry -8.27 rz 25.84 deg; joints [-15.762, 3.559, -16.388, 70.854, -75.702, -333.295]
  MoveL 407 to (-2.18, -100.59, 63.71) mm, rotated rx -159 ry -8.39 rz 25.68 deg; joints [-15.729, 3.524, -16.458, 71.232, -75.342, -333.573]
  MoveL 408 to (-5.22, -99.67, 64.64) mm, rotated rx -157.31 ry -3.23 rz 19.64 deg; joints [-15.671, 3.63, -16.54, 71.222, -78.128, -341.168]
  MoveL 409 to (-4.55, -99.05, 65.14) mm, rotated rx -157.76 ry -3.32 rz 19.55 deg; joints [-15.63, 3.626, -16.624, 71.633, -77.889, -341.393]
  MoveL 410 to (-4.11, -98.25, 65.89) mm, rotated rx -158.38 ry -3.45 rz 19.41 deg; joints [-15.578, 3.582, -16.731, 72.2, -77.538, -341.711]
  MoveL 411 to (-7.39, -97.12, 66.82) mm, rotated rx -156.69 ry 3.53 rz 11.95 deg; joints [-15.54, 3.829, -16.77, 71.378, -81.442, -351.181]
  MoveL 412 to (-7.01, -96.01, 67.92) mm, rotated rx -157.54 ry 3.31 rz 11.73 deg; joints [-15.463, 3.763, -16.921, 72.174, -81.052, -351.577]
  MoveL 413 to (-7, -94.6, 69.39) mm, rotated rx -158.65 ry 2.97 rz 11.41 deg; joints [-15.371, 3.636, -17.112, 73.215, -80.491, -352.129]
  MoveL 414 to (-7.48, -92.8, 71.26) mm, rotated rx -160.01 ry 2.67 rz 10.77 deg; joints [-15.262, 3.451, -17.348, 74.505, -79.854, -353.094]
  MoveL 415 to (-13.13, -89.63, 74.43) mm, rotated rx -159.37 ry 19.94 rz -6.58 deg; joints [-15.239, 4.306, -17.25, 69.785, -89.701, -374.616]
  MoveL 416 to (-11.56, -88.14, 75.37) mm, rotated rx -160.27 ry 19.79 rz -6.94 deg; joints [-15.148, 4.371, -17.444, 70.572, -89.67, -375.094]
  MoveL 417 to (-13.24, -86.21, 77.29) mm, rotated rx -162.24 ry 28.45 rz -16.61 deg; joints [-15.214, 4.82, -17.286, 66.859, -93.953, -386.196]
  MoveL 418 to (-11.92, -86.02, 76.84) mm, rotated rx -162.17 ry 28.58 rz -16.53 deg; joints [-15.224, 4.938, -17.301, 66.771, -94.063, -386.181]
  MoveL 419 to (-10.68, -85.68, 76.53) mm, rotated rx -162.2 ry 28.63 rz -16.49 deg; joints [-15.223, 5.038, -17.334, 66.788, -94.12, -386.188]
  MoveL 420 to (-9.59, -85.18, 76.37) mm, rotated rx -162.32 ry 28.55 rz -16.51 deg; joints [-15.212, 5.11, -17.387, 66.917, -94.088, -386.228]
  MoveL 421 to (-8.43, -83.79, 77.19) mm, rotated rx -163.19 ry 28.35 rz -16.9 deg; joints [-15.132, 5.162, -17.564, 67.623, -94.128, -386.634]
  MoveL 422 to (-8.89, -83.12, 77.86) mm, rotated rx -164.91 ry 32.51 rz -22.2 deg; joints [-15.2, 5.396, -17.434, 65.454, -96.038, -392.222]
  MoveL 423 to (-8.17, -82.86, 77.3) mm, rotated rx -164.78 ry 32.55 rz -22.23 deg; joints [-15.224, 5.452, -17.438, 65.321, -95.958, -392.272]
  MoveL 424 to (-8.66, -82.3, 76.95) mm, rotated rx -164.62 ry 32.03 rz -22.62 deg; joints [-15.244, 5.337, -17.453, 65.339, -95.242, -392.451]
  MoveL 425 to (-8.87, -81.54, 76.84) mm, rotated rx -164.66 ry 31.46 rz -22.94 deg; joints [-15.242, 5.245, -17.508, 65.555, -94.631, -392.594]
  MoveL 426 to (-8.81, -80.61, 76.95) mm, rotated rx -164.86 ry 30.87 rz -23.19 deg; joints [-15.22, 5.176, -17.596, 65.942, -94.124, -392.708]
  MoveL 427 to (-8.67, -79.52, 77.23) mm, rotated rx -165.2 ry 30.2 rz -23.43 deg; joints [-15.183, 5.108, -17.712, 66.479, -93.638, -392.817]
  MoveL 428 to (-8.55, -78.28, 77.67) mm, rotated rx -165.62 ry 29.44 rz -23.68 deg; joints [-15.134, 5.029, -17.851, 67.141, -93.121, -392.938]
  MoveL 429 to (-8.49, -76.94, 78.18) mm, rotated rx -166.09 ry 28.6 rz -23.94 deg; joints [-15.081, 4.938, -18.004, 67.878, -92.57, -393.079]
  MoveL 430 to (-8.51, -75.85, 78.43) mm, rotated rx -165.81 ry 26.24 rz -22.19 deg; joints [-15.019, 4.733, -18.19, 69.315, -91.216, -391.146]
  MoveL 431 to (-8.47, -74.37, 78.86) mm, rotated rx -166.29 ry 25.31 rz -22.34 deg; joints [-14.972, 4.635, -18.36, 70.138, -90.615, -391.216]
  MoveL 432 to (-8.24, -73.1, 79.09) mm, rotated rx -166.67 ry 24.58 rz -22.46 deg; joints [-14.939, 4.574, -18.501, 70.788, -90.141, -391.29]
  MoveL 433 to (-7.81, -72.09, 79.1) mm, rotated rx -166.92 ry 24.08 rz -22.55 deg; joints [-14.922, 4.553, -18.608, 71.229, -89.799, -391.36]
  MoveL 434 to (-6.43, -70.76, 79.48) mm, rotated rx -167.56 ry 23.69 rz -22.28 deg; joints [-14.863, 4.638, -18.793, 72.015, -89.896, -391.231]
  MoveL 435 to (-7.32, -70.96, 78.29) mm, rotated rx -166.81 ry 23.49 rz -22.96 deg; joints [-14.957, 4.51, -18.675, 71.344, -89.033, -391.65]
  MoveL 436 to (-7.42, -70.56, 77.72) mm, rotated rx -166.58 ry 23.18 rz -23.31 deg; joints [-14.993, 4.451, -18.675, 71.246, -88.491, -391.87]
  MoveL 437 to (-6.7, -70.14, 77.26) mm, rotated rx -166 ry 21.5 rz -21.34 deg; joints [-14.989, 4.376, -18.762, 72.008, -87.526, -389.814]
  MoveL 438 to (-5.92, -69.96, 76.53) mm, rotated rx -165.82 ry 21.68 rz -21.42 deg; joints [-15.024, 4.453, -18.75, 71.754, -87.526, -389.898]
  MoveL 439 to (-5.02, -69.82, 75.79) mm, rotated rx -165.64 ry 21.93 rz -21.46 deg; joints [-15.058, 4.549, -18.737, 71.479, -87.597, -389.964]
  MoveL 440 to (-3.99, -69.56, 75.15) mm, rotated rx -165.55 ry 22.14 rz -21.44 deg; joints [-15.082, 4.654, -18.745, 71.312, -87.717, -389.987]
  MoveL 441 to (-2.94, -69.02, 74.77) mm, rotated rx -165.63 ry 22.17 rz -21.34 deg; joints [-15.086, 4.746, -18.799, 71.398, -87.801, -389.959]
  MoveL 442 to (-2.49, -68.6, 74.25) mm, rotated rx -165.54 ry 22.06 rz -21.48 deg; joints [-15.11, 4.765, -18.817, 71.348, -87.59, -390.065]
  MoveL 443 to (-2.05, -68.18, 73.73) mm, rotated rx -165.45 ry 21.96 rz -21.62 deg; joints [-15.134, 4.782, -18.835, 71.298, -87.37, -390.174]
  MoveL 444 to (-1.64, -67.79, 73.2) mm, rotated rx -165.33 ry 21.82 rz -21.74 deg; joints [-15.159, 4.794, -18.85, 71.241, -87.124, -390.251]
  Set speed (50.0 mm/s)
  MoveL 445 to (-1.64, -67.79, 73.2) mm, rotated rx -165.33 ry 21.82 rz -21.74 deg; joints [-15.159, 4.794, -18.85, 71.241, -87.124, -390.251]
  MoveL 446 to (-1.64, -138.5, 143.91) mm, rotated rx -165.33 ry 21.82 rz -21.74 deg; joints [-11.342, 3.915, -14.311, 70.129, -92.08, -387.18]
